Fanuc KAREL source: kc00023.KL

PROGRAM KC00023
%STACKSIZE=65535
%PRIORITY=65535
%NOLOCKGROUP
VAR
I : INTEGER
J : INTEGER
K : INTEGER
R : REAL
B : BOOLEAN
S : STRING[80]
T : STRING[80]
AI : ARRAY[8] OF INTEGER
-- UNRESOLVED DECLARATIONS (source type spelling not recovered)
-- P : TYPE_0x001F (type_u16=0x001F)
-- Q : TYPE_0x001F (type_u16=0x001F)
-- AB : ARRAY[244] OF TYPE_0x0018 (type_u16=0x2018)
ROUTINE BUMP(P1 : INTEGER) FROM KC00023
ROUTINE BUMP
BEGIN
P1=(P1 + 1)
END BUMP
BEGIN
S=''
T='I'
-- UNSAFE_SOURCE_IR line 22: BUMP(ARG_1_UNRESOLVED)
END KC00023
